// TIA Portal V20 export
DATA_BLOCK "DB_CycleStartStop"   // DB81
// stored: InstanceOfName FB_CycleStartStop, InstanceOfType FB
"FB_CycleStartStop"
   // VAR
   //    sChan1Start : Bool;
   //    sResquestStopNextCycle : Bool;
   //    sTimePowerSupplyAlarm : TON_TIME;
   //    sRT_CNAskStopCycle : R_TRIG;
   // END_VAR
BEGIN
END_DATA_BLOCK
